{attribute 'qualified_only'}
{attribute 'strict'}
{attribute 'to_string'}
TYPE eSlideposition :
(
	In := 0,
	Out:=1,
	Unknown:=2
);
END_TYPE

(* stored: Version 1.1.0.1
   DUT eSlideposition: Id {09da7d7e-cdca-4849-b3cf-aebb22604c21} *)
